% RSLogix 500 project counter2.RSS, saved by version 8.30.00.16 %
PROJECT "UNTITLED"    % processor: Bul.1763 MicroLogix 1100 Series B %

PROGRAM FILES
  LAD 2   5 rungs

DATA FILES
  O0 OUTPUT  4 elements
  I1 INPUT  6 elements
  S2 STATUS  66 elements
  B3 BINARY  1 elements
  T4 TIMER  1 elements
  C5 COUNTER  1 elements
  R6 CONTROL  1 elements
  N7 INTEGER  1 elements
  F8 FLOAT  1 elements

LADDER 2
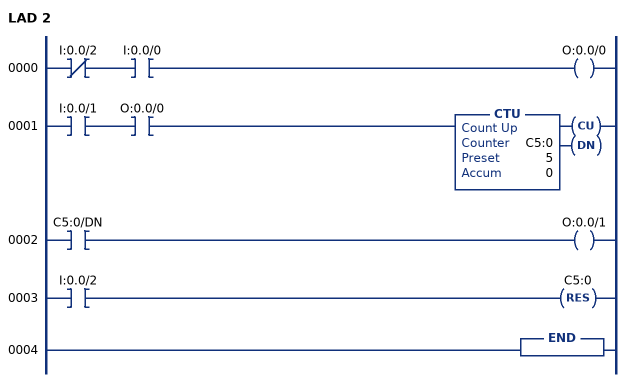
% Rung: 0 %
SOR XIO I:0.0/2 XIC I:0.0/0 OTE O:0.0/0 EOR
% Rung: 1 %
SOR XIC I:0.0/1 XIC O:0.0/0 CTU C5:0 5 0 EOR
% Rung: 2 %
SOR XIC C5:0/DN OTE O:0.0/1 EOR
% Rung: 3 %
SOR XIC I:0.0/2 RES C5:0 EOR
% Rung: 4 %
SOR END EOR

DATA TABLE (non-zero values as saved)
DATA C5
% .PRE .ACC %
% C5:0 % 5 0
